// TIA Portal V17 export
DATA_BLOCK "MotorInst"   // DB200
// Background instance of FB_Motor
// stored: OfType FB_Motor
BEGIN
END_DATA_BLOCK
